ABB RobotStudio station: Solution_20180910-123525.rsstn

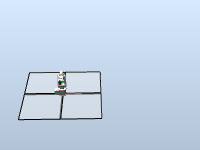
Station Solution3 (saved by RobotStudio 6.7.7936.1011)
Controller MTRN4230
  mechanical unit ROB_1: IRB120_3_58__01, 6 joints, base frame (0, 0, 0) mm
Layout (positions relative to the parent item):
  - IRB120_3_58__01 [mechanism, from Robots\IRB120_3_58_G_01.rslib] at (0, 0, 0) mm; joint values [-1.5708, 0, 0, 0, 0, 0] (rad or m)
